{attribute 'GeneratedUsingTerminal: EK1100-0000-0018'}
{attribute addProperty BoxType "EK1100-0000-0018"}
{attribute addProperty Id "Beckhoff_EL33xxEK1122Beckhoff_EL33xxEK1122_F347A86E2A_0001_EL3311_0000_0016EL3311_768B3E6721A_0002_EL3311_0000_0017EL3311_768B3E6721A_0003_EL3311_0000_0018EL3311_2A8D498221A_0004_EL3311_0000_0019EL3311_2A8D498221A_0005_EL3311_0000_0020EL3311_2A8D498221A_0006_EL3311_0000_0021EL3311_2A8D498221A_0007_EL3311_0000_0022EL3311_2A8D498221A_0008_EL3311_0000_0023EL3311_2A8D498221A_0009_EL3312_0000_0016EL3312_4865548330A_0010_EL3312_0000_0017EL3312_4865548330A_0011_EL3312_0000_0018EL3312_792163DD30A_0012_EL3312_0000_0019EL3312_792163DD30A_0013_EL3312_0000_0020EL3312_792163DD30A_0014_EL3312_0000_0021EL3312_792163DD30A_0015_EL3312_0000_0022EL3312_792163DD30A_0016_EL3312_0000_0023EL3312_792163DD30A_0017_EL3314_0000_0016EL3314_18BBAF4748A_0018_EL3314_0000_0017EL3314_18BBAF4748A_0019_EL3314_0000_0018EL3314_B654D23048A_0020_EL3314_0000_0019EL3314_B654D23048A_0021_EL3314_0000_0020EL3314_B654D23048A_0022_EL3314_0000_0021EL3314_B654D23048A_0023_EL3314_0000_0022EL3314_B654D23048A_0024_EL3314_0000_0023EL3314_B654D23048A_0025_EL3314_0000_0024EL3314_B654D23048A_0026_EL3314_0002_0016EL3314_6E4DFFE556A_0027_EL3314_0010_0016EL3314_C9476E1C48A_0028_EL3314_0010_0017EL3314_C9476E1C48A_0029_EL3314_0010_0018EL3314_C9476E1C48A_0030_EL3314_0010_0019EL3314_C9476E1C48A_0031_EL3314_0010_0020EL3314_C9476E1C48A_0032_EL3314_0010_0021EL3314_C9476E1C48A_0033_EL3314_0090_0016EL3314_B654D23048A_0034_EL3314_0090_0017EL3314_B654D23048A_0035_EL3318_0000_0016EL3318_44C149FC68A_0036_EL3318_0000_0017EL3318_44C149FC68A_0037_EL3318_0000_0018EL3318_44C149FC68A_0038_EL3318_0000_0019EL3318_44C149FC68A_0039_EL3318_0000_0020EL3318_44C149FC68A_0040_EL3318_0000_0021EL3318_44C149FC68A_0041_EL3318_0000_0022EL3318_44C149FC68A_0042_EL3351_0000_0016EL3351_6847F28330A_0043_EL3351_0000_0017EL3351_6847F28330A_0044_EL3351_0000_0018EL3351_6847F28330A_0045_EL3351_0000_0019EL3351_6847F28330A_0046_EL3351_0000_0020EL3351_6847F28330A_0047_EL3356_0000_0017EL3356_8E3EBEA027A_0048_EL3356_0000_0018EL3356_8E3EBEA027A_0049_EL3356_0000_0019EL3356_8E3EBEA027A_0050_EL3356_0000_0020EL3356_8E3EBEA027A_0051_EL3356_0000_0021EL3356_8E3EBEA027A_0052_EL3356_0000_0022EL3356_8E3EBEA027A_0053_EL3356_0000_0023EL3356_8E3EBEA027A_0054_EL3356_0000_0024EL3356_8E3EBEA027A_0055_EL3356_0000_0025EL3356_8E3EBEA027A_0056_EL3356_0010_0017EL3356_1EAAA6FF28A_0057_EL3356_0010_0018EL3356_1EAAA6FF28A_0058_EL3356_0010_0019EL3356_1EAAA6FF28A_0059_EL3356_0010_0020EL3356_1EAAA6FF28A_0060_EL3356_0010_0021EL3356_1EAAA6FF28A_0061_EL3356_0010_0022EL3356_1EAAA6FF28A_0062_EL3356_0010_0023EL3356_1EAAA6FF28A_0063_EL3356_0010_0024EL3356_1EAAA6FF28A_0064_EL3356_0010_0025EL3356_1EAAA6FF28A_0065_EL3356_0020_0025EL3356_1EAAA6FF28A_0066_EL3356_0090_0025EL3356_1EAAA6FF28"}
{attribute addProperty CRC "2001989952"}
{attribute addProperty Size "2459"}
TYPE Beckhoff_EL33xx_7753F140 EXTENDS EK1100_1FC0878B :
STRUCT
	{attribute addProperty Name "Beckhoff_EL33xxEK1122"}
	{attribute addProperty PreviousPort "Beckhoff EL33xx : B"}
	Beckhoff_EL33xxEK1122 : Beckhoff_EL33xxEK1122_F347A86E;
	{attribute addProperty Name "A_0001_EL3311_0000_0016"}
	{attribute addProperty PreviousPort "Beckhoff EL33xxEK1122 : C"}
	A_0001_EL3311_0000_0016 : EL3311_768B3E67;
	{attribute addProperty Name "A_0002_EL3311_0000_0017"}
	{attribute addProperty PreviousPort "A_0001(EL3311-0000-0016) : B"}
	A_0002_EL3311_0000_0017 : EL3311_768B3E67;
	{attribute addProperty Name "A_0003_EL3311_0000_0018"}
	{attribute addProperty PreviousPort "A_0002(EL3311-0000-0017) : B"}
	A_0003_EL3311_0000_0018 : EL3311_2A8D4982;
	{attribute addProperty Name "A_0004_EL3311_0000_0019"}
	{attribute addProperty PreviousPort "A_0003(EL3311-0000-0018) : B"}
	A_0004_EL3311_0000_0019 : EL3311_2A8D4982;
	{attribute addProperty Name "A_0005_EL3311_0000_0020"}
	{attribute addProperty PreviousPort "A_0004(EL3311-0000-0019) : B"}
	A_0005_EL3311_0000_0020 : EL3311_2A8D4982;
	{attribute addProperty Name "A_0006_EL3311_0000_0021"}
	{attribute addProperty PreviousPort "A_0005(EL3311-0000-0020) : B"}
	A_0006_EL3311_0000_0021 : EL3311_2A8D4982;
	{attribute addProperty Name "A_0007_EL3311_0000_0022"}
	{attribute addProperty PreviousPort "A_0006(EL3311-0000-0021) : B"}
	A_0007_EL3311_0000_0022 : EL3311_2A8D4982;
	{attribute addProperty Name "A_0008_EL3311_0000_0023"}
	{attribute addProperty PreviousPort "A_0007(EL3311-0000-0022) : B"}
	A_0008_EL3311_0000_0023 : EL3311_2A8D4982;
	{attribute addProperty Name "A_0009_EL3312_0000_0016"}
	{attribute addProperty PreviousPort "A_0008(EL3311-0000-0023) : B"}
	A_0009_EL3312_0000_0016 : EL3312_48655483;
	{attribute addProperty Name "A_0010_EL3312_0000_0017"}
	{attribute addProperty PreviousPort "A_0009(EL3312-0000-0016) : B"}
	A_0010_EL3312_0000_0017 : EL3312_48655483;
	{attribute addProperty Name "A_0011_EL3312_0000_0018"}
	{attribute addProperty PreviousPort "A_0010(EL3312-0000-0017) : B"}
	A_0011_EL3312_0000_0018 : EL3312_792163DD;
	{attribute addProperty Name "A_0012_EL3312_0000_0019"}
	{attribute addProperty PreviousPort "A_0011(EL3312-0000-0018) : B"}
	A_0012_EL3312_0000_0019 : EL3312_792163DD;
	{attribute addProperty Name "A_0013_EL3312_0000_0020"}
	{attribute addProperty PreviousPort "A_0012(EL3312-0000-0019) : B"}
	A_0013_EL3312_0000_0020 : EL3312_792163DD;
	{attribute addProperty Name "A_0014_EL3312_0000_0021"}
	{attribute addProperty PreviousPort "A_0013(EL3312-0000-0020) : B"}
	A_0014_EL3312_0000_0021 : EL3312_792163DD;
	{attribute addProperty Name "A_0015_EL3312_0000_0022"}
	{attribute addProperty PreviousPort "A_0014(EL3312-0000-0021) : B"}
	A_0015_EL3312_0000_0022 : EL3312_792163DD;
	{attribute addProperty Name "A_0016_EL3312_0000_0023"}
	{attribute addProperty PreviousPort "A_0015(EL3312-0000-0022) : B"}
	A_0016_EL3312_0000_0023 : EL3312_792163DD;
	{attribute addProperty Name "A_0017_EL3314_0000_0016"}
	{attribute addProperty PreviousPort "A_0016(EL3312-0000-0023) : B"}
	A_0017_EL3314_0000_0016 : EL3314_18BBAF47;
	{attribute addProperty Name "A_0018_EL3314_0000_0017"}
	{attribute addProperty PreviousPort "A_0017(EL3314-0000-0016) : B"}
	A_0018_EL3314_0000_0017 : EL3314_18BBAF47;
	{attribute addProperty Name "A_0019_EL3314_0000_0018"}
	{attribute addProperty PreviousPort "A_0018(EL3314-0000-0017) : B"}
	A_0019_EL3314_0000_0018 : EL3314_B654D230;
	{attribute addProperty Name "A_0020_EL3314_0000_0019"}
	{attribute addProperty PreviousPort "A_0019(EL3314-0000-0018) : B"}
	A_0020_EL3314_0000_0019 : EL3314_B654D230;
	{attribute addProperty Name "A_0021_EL3314_0000_0020"}
	{attribute addProperty PreviousPort "A_0020(EL3314-0000-0019) : B"}
	A_0021_EL3314_0000_0020 : EL3314_B654D230;
	{attribute addProperty Name "A_0022_EL3314_0000_0021"}
	{attribute addProperty PreviousPort "A_0021(EL3314-0000-0020) : B"}
	A_0022_EL3314_0000_0021 : EL3314_B654D230;
	{attribute addProperty Name "A_0023_EL3314_0000_0022"}
	{attribute addProperty PreviousPort "A_0022(EL3314-0000-0021) : B"}
	A_0023_EL3314_0000_0022 : EL3314_B654D230;
	{attribute addProperty Name "A_0024_EL3314_0000_0023"}
	{attribute addProperty PreviousPort "A_0023(EL3314-0000-0022) : B"}
	A_0024_EL3314_0000_0023 : EL3314_B654D230;
	{attribute addProperty Name "A_0025_EL3314_0000_0024"}
	{attribute addProperty PreviousPort "A_0024(EL3314-0000-0023) : B"}
	A_0025_EL3314_0000_0024 : EL3314_B654D230;
	{attribute addProperty Name "A_0026_EL3314_0002_0016"}
	{attribute addProperty PreviousPort "A_0025(EL3314-0000-0024) : B"}
	A_0026_EL3314_0002_0016 : EL3314_6E4DFFE5;
	{attribute addProperty Name "A_0027_EL3314_0010_0016"}
	{attribute addProperty PreviousPort "A_0026(EL3314-0002-0016) : B"}
	A_0027_EL3314_0010_0016 : EL3314_C9476E1C;
	{attribute addProperty Name "A_0028_EL3314_0010_0017"}
	{attribute addProperty PreviousPort "A_0027(EL3314-0010-0016) : B"}
	A_0028_EL3314_0010_0017 : EL3314_C9476E1C;
	{attribute addProperty Name "A_0029_EL3314_0010_0018"}
	{attribute addProperty PreviousPort "A_0028(EL3314-0010-0017) : B"}
	A_0029_EL3314_0010_0018 : EL3314_C9476E1C;
	{attribute addProperty Name "A_0030_EL3314_0010_0019"}
	{attribute addProperty PreviousPort "A_0029(EL3314-0010-0018) : B"}
	A_0030_EL3314_0010_0019 : EL3314_C9476E1C;
	{attribute addProperty Name "A_0031_EL3314_0010_0020"}
	{attribute addProperty PreviousPort "A_0030(EL3314-0010-0019) : B"}
	A_0031_EL3314_0010_0020 : EL3314_C9476E1C;
	{attribute addProperty Name "A_0032_EL3314_0010_0021"}
	{attribute addProperty PreviousPort "A_0031(EL3314-0010-0020) : B"}
	A_0032_EL3314_0010_0021 : EL3314_C9476E1C;
	{attribute addProperty Name "A_0033_EL3314_0090_0016"}
	{attribute addProperty PreviousPort "A_0032(EL3314-0010-0021) : B"}
	A_0033_EL3314_0090_0016 : EL3314_B654D230;
	{attribute addProperty Name "A_0034_EL3314_0090_0017"}
	{attribute addProperty PreviousPort "A_0033(EL3314-0090-0016) : B"}
	A_0034_EL3314_0090_0017 : EL3314_B654D230;
	{attribute addProperty Name "A_0035_EL3318_0000_0016"}
	{attribute addProperty PreviousPort "A_0034(EL3314-0090-0017) : B"}
	A_0035_EL3318_0000_0016 : EL3318_44C149FC;
	{attribute addProperty Name "A_0036_EL3318_0000_0017"}
	{attribute addProperty PreviousPort "A_0035(EL3318-0000-0016) : B"}
	A_0036_EL3318_0000_0017 : EL3318_44C149FC;
	{attribute addProperty Name "A_0037_EL3318_0000_0018"}
	{attribute addProperty PreviousPort "A_0036(EL3318-0000-0017) : B"}
	A_0037_EL3318_0000_0018 : EL3318_44C149FC;
	{attribute addProperty Name "A_0038_EL3318_0000_0019"}
	{attribute addProperty PreviousPort "A_0037(EL3318-0000-0018) : B"}
	A_0038_EL3318_0000_0019 : EL3318_44C149FC;
	{attribute addProperty Name "A_0039_EL3318_0000_0020"}
	{attribute addProperty PreviousPort "A_0038(EL3318-0000-0019) : B"}
	A_0039_EL3318_0000_0020 : EL3318_44C149FC;
	{attribute addProperty Name "A_0040_EL3318_0000_0021"}
	{attribute addProperty PreviousPort "A_0039(EL3318-0000-0020) : B"}
	A_0040_EL3318_0000_0021 : EL3318_44C149FC;
	{attribute addProperty Name "A_0041_EL3318_0000_0022"}
	{attribute addProperty PreviousPort "A_0040(EL3318-0000-0021) : B"}
	A_0041_EL3318_0000_0022 : EL3318_44C149FC;
	{attribute addProperty Name "A_0042_EL3351_0000_0016"}
	{attribute addProperty PreviousPort "A_0041(EL3318-0000-0022) : B"}
	A_0042_EL3351_0000_0016 : EL3351_6847F283;
	{attribute addProperty Name "A_0043_EL3351_0000_0017"}
	{attribute addProperty PreviousPort "A_0042(EL3351-0000-0016) : B"}
	A_0043_EL3351_0000_0017 : EL3351_6847F283;
	{attribute addProperty Name "A_0044_EL3351_0000_0018"}
	{attribute addProperty PreviousPort "A_0043(EL3351-0000-0017) : B"}
	A_0044_EL3351_0000_0018 : EL3351_6847F283;
	{attribute addProperty Name "A_0045_EL3351_0000_0019"}
	{attribute addProperty PreviousPort "A_0044(EL3351-0000-0018) : B"}
	A_0045_EL3351_0000_0019 : EL3351_6847F283;
	{attribute addProperty Name "A_0046_EL3351_0000_0020"}
	{attribute addProperty PreviousPort "A_0045(EL3351-0000-0019) : B"}
	A_0046_EL3351_0000_0020 : EL3351_6847F283;
	{attribute addProperty Name "A_0047_EL3356_0000_0017"}
	{attribute addProperty PreviousPort "A_0046(EL3351-0000-0020) : B"}
	A_0047_EL3356_0000_0017 : EL3356_8E3EBEA0;
	{attribute addProperty Name "A_0048_EL3356_0000_0018"}
	{attribute addProperty PreviousPort "A_0047(EL3356-0000-0017) : B"}
	A_0048_EL3356_0000_0018 : EL3356_8E3EBEA0;
	{attribute addProperty Name "A_0049_EL3356_0000_0019"}
	{attribute addProperty PreviousPort "A_0048(EL3356-0000-0018) : B"}
	A_0049_EL3356_0000_0019 : EL3356_8E3EBEA0;
	{attribute addProperty Name "A_0050_EL3356_0000_0020"}
	{attribute addProperty PreviousPort "A_0049(EL3356-0000-0019) : B"}
	A_0050_EL3356_0000_0020 : EL3356_8E3EBEA0;
	{attribute addProperty Name "A_0051_EL3356_0000_0021"}
	{attribute addProperty PreviousPort "A_0050(EL3356-0000-0020) : B"}
	A_0051_EL3356_0000_0021 : EL3356_8E3EBEA0;
	{attribute addProperty Name "A_0052_EL3356_0000_0022"}
	{attribute addProperty PreviousPort "A_0051(EL3356-0000-0021) : B"}
	A_0052_EL3356_0000_0022 : EL3356_8E3EBEA0;
	{attribute addProperty Name "A_0053_EL3356_0000_0023"}
	{attribute addProperty PreviousPort "A_0052(EL3356-0000-0022) : B"}
	A_0053_EL3356_0000_0023 : EL3356_8E3EBEA0;
	{attribute addProperty Name "A_0054_EL3356_0000_0024"}
	{attribute addProperty PreviousPort "A_0053(EL3356-0000-0023) : B"}
	A_0054_EL3356_0000_0024 : EL3356_8E3EBEA0;
	{attribute addProperty Name "A_0055_EL3356_0000_0025"}
	{attribute addProperty PreviousPort "A_0054(EL3356-0000-0024) : B"}
	A_0055_EL3356_0000_0025 : EL3356_8E3EBEA0;
	{attribute addProperty Name "A_0056_EL3356_0010_0017"}
	{attribute addProperty PreviousPort "A_0055(EL3356-0000-0025) : B"}
	A_0056_EL3356_0010_0017 : EL3356_1EAAA6FF;
	{attribute addProperty Name "A_0057_EL3356_0010_0018"}
	{attribute addProperty PreviousPort "A_0056(EL3356-0010-0017) : B"}
	A_0057_EL3356_0010_0018 : EL3356_1EAAA6FF;
	{attribute addProperty Name "A_0058_EL3356_0010_0019"}
	{attribute addProperty PreviousPort "A_0057(EL3356-0010-0018) : B"}
	A_0058_EL3356_0010_0019 : EL3356_1EAAA6FF;
	{attribute addProperty Name "A_0059_EL3356_0010_0020"}
	{attribute addProperty PreviousPort "A_0058(EL3356-0010-0019) : B"}
	A_0059_EL3356_0010_0020 : EL3356_1EAAA6FF;
	{attribute addProperty Name "A_0060_EL3356_0010_0021"}
	{attribute addProperty PreviousPort "A_0059(EL3356-0010-0020) : B"}
	A_0060_EL3356_0010_0021 : EL3356_1EAAA6FF;
	{attribute addProperty Name "A_0061_EL3356_0010_0022"}
	{attribute addProperty PreviousPort "A_0060(EL3356-0010-0021) : B"}
	A_0061_EL3356_0010_0022 : EL3356_1EAAA6FF;
	{attribute addProperty Name "A_0062_EL3356_0010_0023"}
	{attribute addProperty PreviousPort "A_0061(EL3356-0010-0022) : B"}
	A_0062_EL3356_0010_0023 : EL3356_1EAAA6FF;
	{attribute addProperty Name "A_0063_EL3356_0010_0024"}
	{attribute addProperty PreviousPort "A_0062(EL3356-0010-0023) : B"}
	A_0063_EL3356_0010_0024 : EL3356_1EAAA6FF;
	{attribute addProperty Name "A_0064_EL3356_0010_0025"}
	{attribute addProperty PreviousPort "A_0063(EL3356-0010-0024) : B"}
	A_0064_EL3356_0010_0025 : EL3356_1EAAA6FF;
	{attribute addProperty Name "A_0065_EL3356_0020_0025"}
	{attribute addProperty PreviousPort "A_0064(EL3356-0010-0025) : B"}
	A_0065_EL3356_0020_0025 : EL3356_1EAAA6FF;
	{attribute addProperty Name "A_0066_EL3356_0090_0025"}
	{attribute addProperty PreviousPort "A_0065(EL3356-0020-0025) : B"}
	A_0066_EL3356_0090_0025 : EL3356_1EAAA6FF;
END_STRUCT
END_TYPE

(* stored: Version 1.2.0.0, ProductVersion 3.1.4024.9
   DUT Beckhoff_EL33xx_7753F140: Id {ca0495be-b78d-44bc-a1dd-5676f8fe77f1} *)
